FUNCTION_BLOCK F_RND (* rounds a real down to n digits total, round(3.1415,2) = 3.1 *)
  (* Standard: OSCAT; Classification: Math *)
  (* Version 0.0, 2011-07-21, 4DIAC-IDE, 4DIAC-Consortium *)
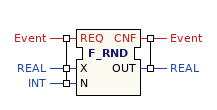
  EVENT_INPUT
    REQ WITH X, N; (* Service Request *)
  END_EVENT
  EVENT_OUTPUT
    CNF WITH OUT; (* Confirmation of Requested Service *)
  END_EVENT
  VAR_INPUT
    X : REAL; (* Input for round *)
    N : INT; (* Digits behind comma *)
  END_VAR
  VAR_OUTPUT
    OUT : REAL; (* Round outcome *)
  END_VAR
END_FUNCTION_BLOCK
